Omron CX-Programmer project NewProject (CX-Programmer 9.75)

# PLC NewPLC1: CQM1 CPU43

## Program NewProgram1 (no task)

### Section Section1

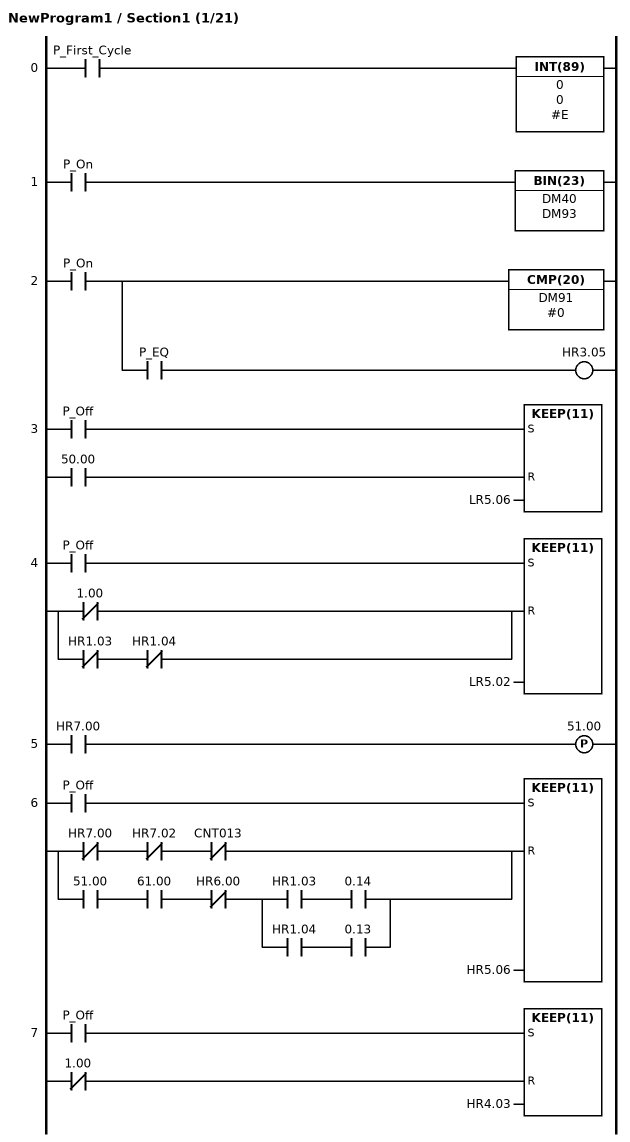
; rung 0
LD P_First_Cycle
INT(89) 0 0 #E
; rung 1
LD P_On
BIN(23) DM40 DM93
; rung 2
LD P_On
CMP(20) DM91 #0
AND P_EQ
OUT HR3.05
; rung 3
LD P_Off
LD 50.00
KEEP(11) LR5.06
; rung 4
LD P_Off
LDNOT 1.00
LDNOT HR1.03
ANDNOT HR1.04
ORLD
KEEP(11) LR5.02
; rung 5
LD HR7.00
DIFU(13) 51.00
; rung 6
LD P_Off
LDNOT HR7.00
ANDNOT HR7.02
ANDNOT CNT013
LD 51.00
AND 61.00
ANDNOT HR6.00
LD HR1.03
AND 0.14
LD HR1.04
AND 0.13
ORLD
ANDLD
ORLD
KEEP(11) HR5.06
; rung 7
LD P_Off
LDNOT 1.00
KEEP(11) HR4.03

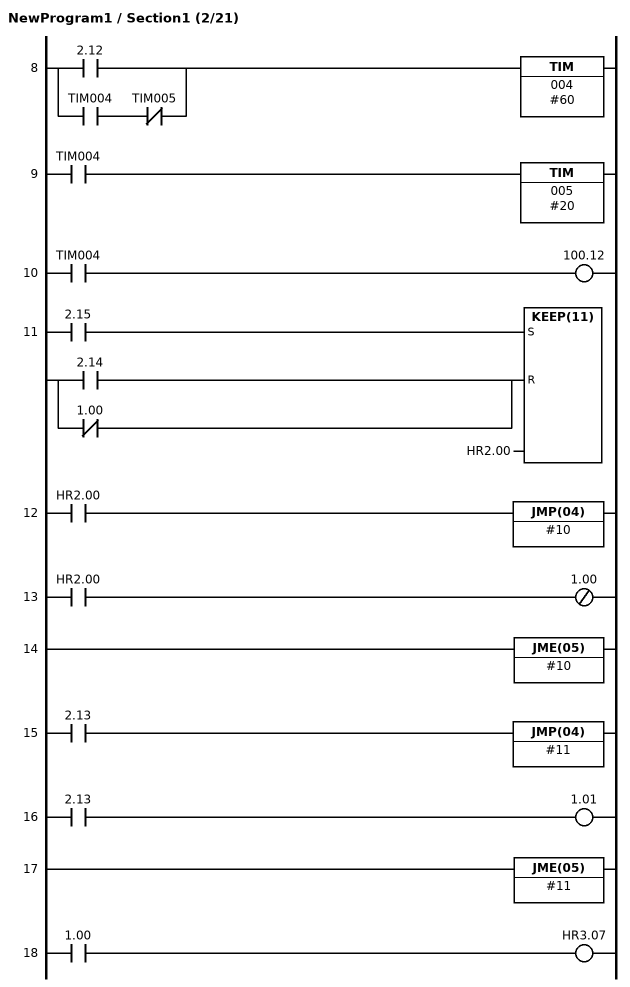
; rung 8
LD 2.12
LD TIM004
ANDNOT TIM005
ORLD
TIM 004 #60
; rung 9
LD TIM004
TIM 005 #20
; rung 10
LD TIM004
OUT 100.12
; rung 11
LD 2.15
LD 2.14
ORNOT 1.00
KEEP(11) HR2.00
; rung 12
LD HR2.00
JMP(04) #10
; rung 13
LD HR2.00
OUTNOT 1.00
; rung 14
JME(05) #10
; rung 15
LD 2.13
JMP(04) #11
; rung 16
LD 2.13
OUT 1.01
; rung 17
JME(05) #11
; rung 18
LD 1.00
OUT HR3.07

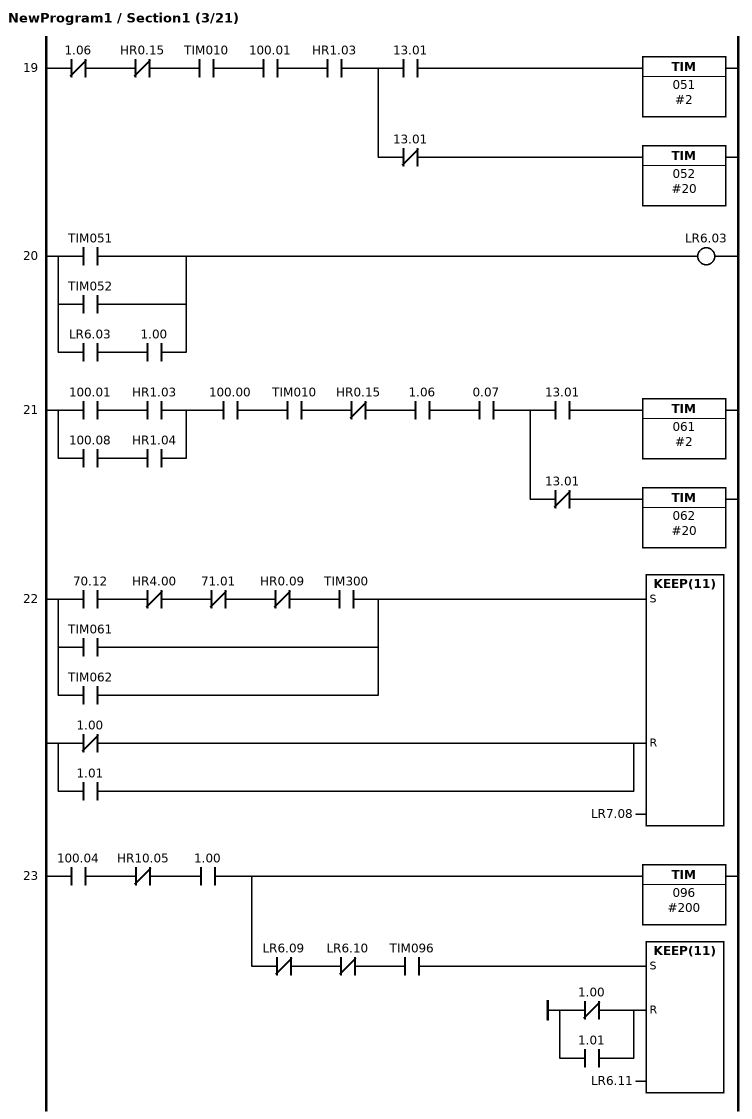
; rung 19
LDNOT 1.06
ANDNOT HR0.15
AND TIM010
AND 100.01
AND HR1.03
OUT TR0
AND 13.01
TIM 051 #2
LD TR0
ANDNOT 13.01
TIM 052 #20
; rung 20
LD TIM051
OR TIM052
LD LR6.03
AND 1.00
ORLD
OUT LR6.03
; rung 21
LD 100.01
AND HR1.03
LD 100.08
AND HR1.04
ORLD
AND 100.00
AND TIM010
ANDNOT HR0.15
AND 1.06
AND 0.07
OUT TR0
AND 13.01
TIM 061 #2
LD TR0
ANDNOT 13.01
TIM 062 #20
; rung 22
LD 70.12
ANDNOT HR4.00
ANDNOT 71.01
ANDNOT HR0.09
AND TIM300
OR TIM061
OR TIM062
LDNOT 1.00
OR 1.01
KEEP(11) LR7.08
; rung 23
LD 100.04
ANDNOT HR10.05
AND 1.00
TIM 096 #200
ANDNOT LR6.09
ANDNOT LR6.10
AND TIM096
LDNOT 1.00
OR 1.01
KEEP(11) LR6.11

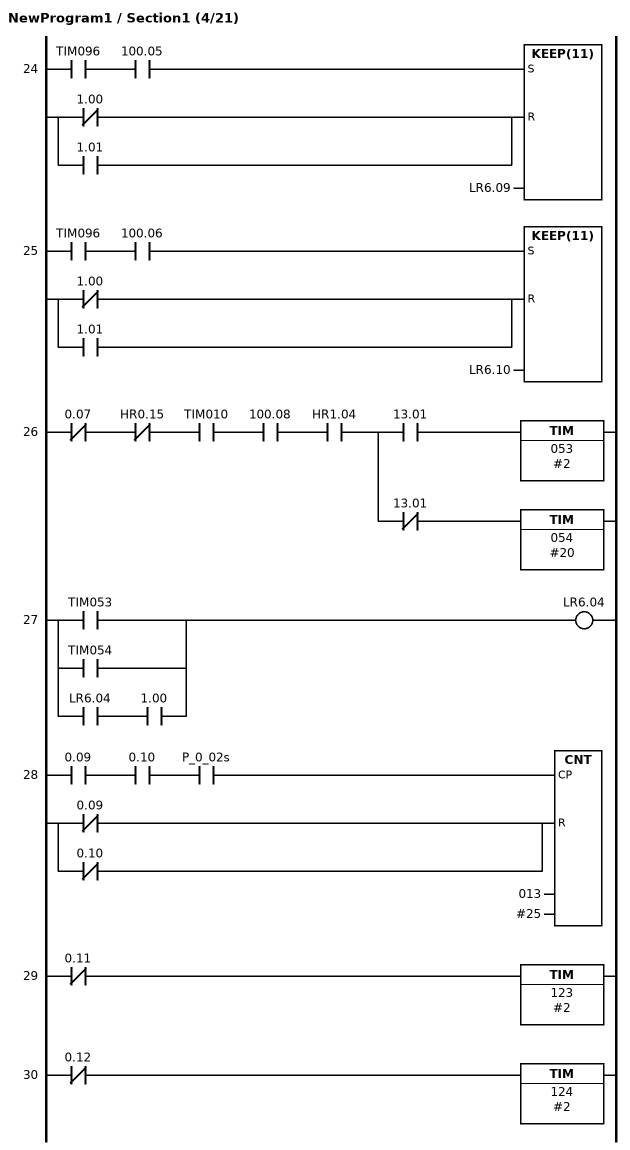
; rung 24
LD TIM096
AND 100.05
LDNOT 1.00
OR 1.01
KEEP(11) LR6.09
; rung 25
LD TIM096
AND 100.06
LDNOT 1.00
OR 1.01
KEEP(11) LR6.10
; rung 26
LDNOT 0.07
ANDNOT HR0.15
AND TIM010
AND 100.08
AND HR1.04
OUT TR0
AND 13.01
TIM 053 #2
LD TR0
ANDNOT 13.01
TIM 054 #20
; rung 27
LD TIM053
OR TIM054
LD LR6.04
AND 1.00
ORLD
OUT LR6.04
; rung 28
LD 0.09
AND 0.10
AND P_0_02s
LDNOT 0.09
ORNOT 0.10
CNT 013 #25
; rung 29
LDNOT 0.11
TIM 123 #2
; rung 30
LDNOT 0.12
TIM 124 #2

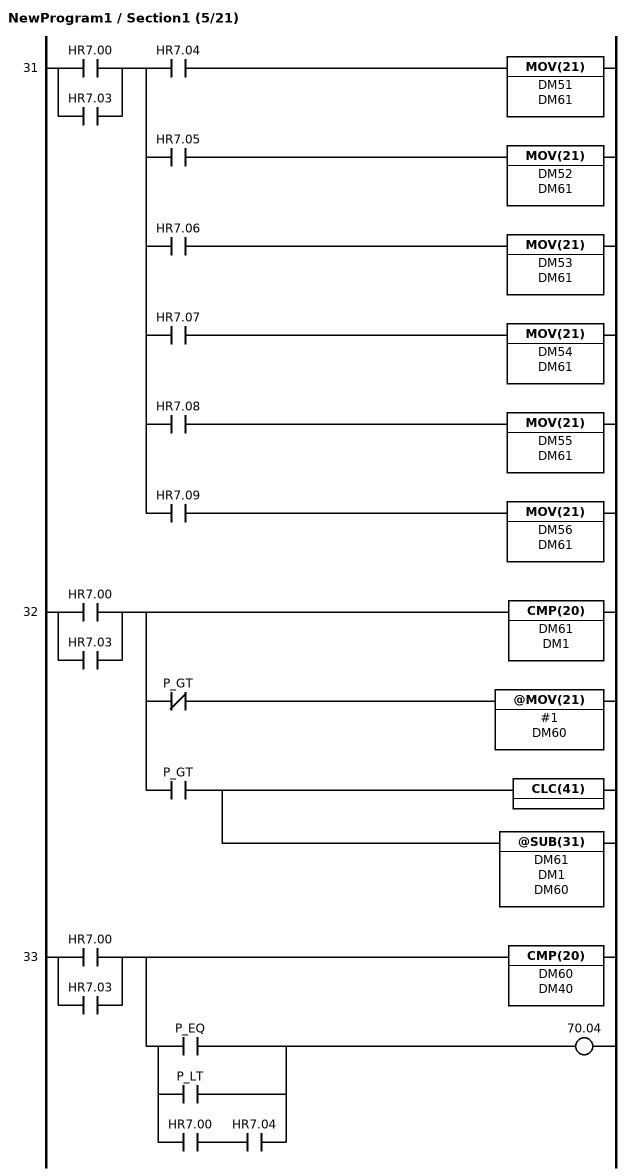
; rung 31
LD HR7.00
OR HR7.03
OUT TR0
AND HR7.04
MOV(21) DM51 DM61
LD TR0
AND HR7.05
MOV(21) DM52 DM61
LD TR0
AND HR7.06
MOV(21) DM53 DM61
LD TR0
AND HR7.07
MOV(21) DM54 DM61
LD TR0
AND HR7.08
MOV(21) DM55 DM61
LD TR0
AND HR7.09
MOV(21) DM56 DM61
; rung 32
LD HR7.00
OR HR7.03
OUT TR0
CMP(20) DM61 DM1
ANDNOT P_GT
@MOV(21) #1 DM60
LD TR0
AND P_GT
CLC(41)
@SUB(31) DM61 DM1 DM60
; rung 33
LD HR7.00
OR HR7.03
CMP(20) DM60 DM40
LD P_EQ
OR P_LT
LD HR7.00
AND HR7.04
ORLD
ANDLD
OUT 70.04

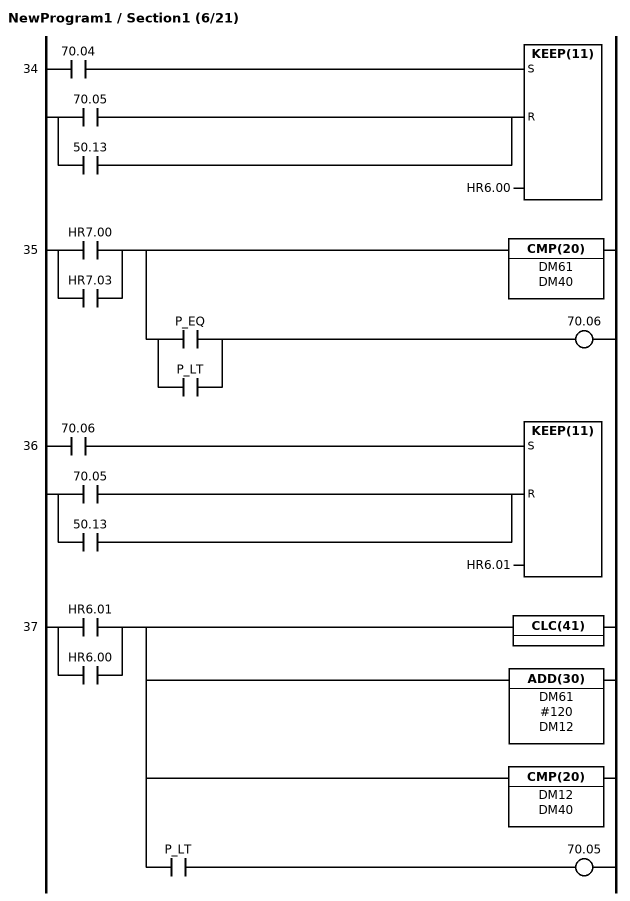
; rung 34
LD 70.04
LD 70.05
OR 50.13
KEEP(11) HR6.00
; rung 35
LD HR7.00
OR HR7.03
CMP(20) DM61 DM40
LD P_EQ
OR P_LT
ANDLD
OUT 70.06
; rung 36
LD 70.06
LD 70.05
OR 50.13
KEEP(11) HR6.01
; rung 37
LD HR6.01
OR HR6.00
CLC(41)
ADD(30) DM61 #120 DM12
CMP(20) DM12 DM40
AND P_LT
OUT 70.05

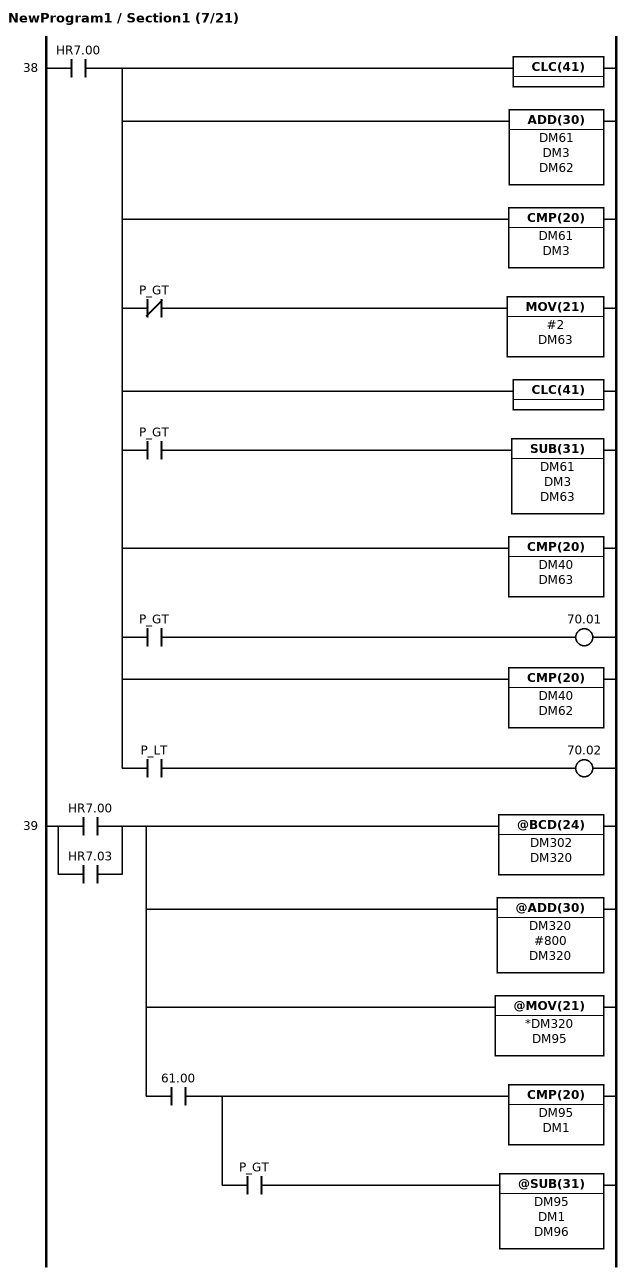
; rung 38
LD HR7.00
OUT TR0
CLC(41)
ADD(30) DM61 DM3 DM62
CMP(20) DM61 DM3
ANDNOT P_GT
MOV(21) #2 DM63
LD TR0
CLC(41)
AND P_GT
SUB(31) DM61 DM3 DM63
LD TR0
CMP(20) DM40 DM63
AND P_GT
OUT 70.01
LD TR0
CMP(20) DM40 DM62
AND P_LT
OUT 70.02
; rung 39
LD HR7.00
OR HR7.03
@BCD(24) DM302 DM320
@ADD(30) DM320 #800 DM320
@MOV(21) *DM320 DM95
AND 61.00
CMP(20) DM95 DM1
AND P_GT
@SUB(31) DM95 DM1 DM96

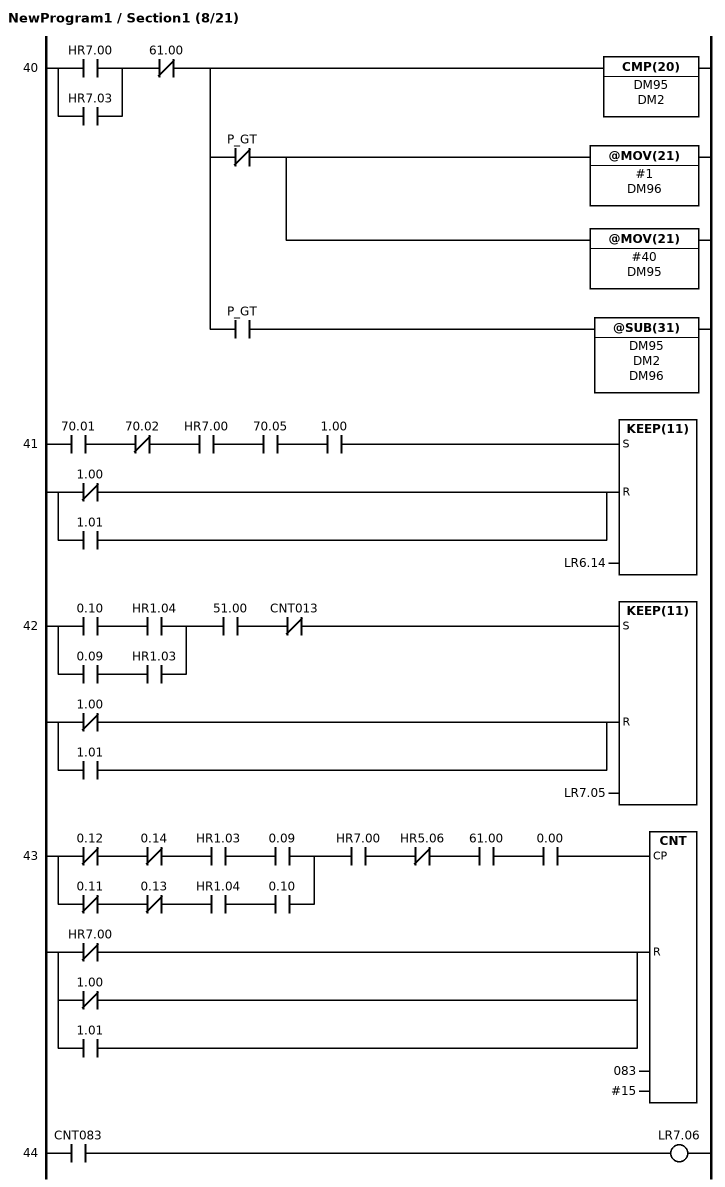
; rung 40
LD HR7.00
OR HR7.03
ANDNOT 61.00
OUT TR0
CMP(20) DM95 DM2
ANDNOT P_GT
@MOV(21) #1 DM96
@MOV(21) #40 DM95
LD TR0
AND P_GT
@SUB(31) DM95 DM2 DM96
; rung 41
LD 70.01
ANDNOT 70.02
AND HR7.00
AND 70.05
AND 1.00
LDNOT 1.00
OR 1.01
KEEP(11) LR6.14
; rung 42
LD 0.10
AND HR1.04
LD 0.09
AND HR1.03
ORLD
AND 51.00
ANDNOT CNT013
LDNOT 1.00
OR 1.01
KEEP(11) LR7.05
; rung 43
LDNOT 0.12
ANDNOT 0.14
AND HR1.03
AND 0.09
LDNOT 0.11
ANDNOT 0.13
AND HR1.04
AND 0.10
ORLD
AND HR7.00
ANDNOT HR5.06
AND 61.00
AND 0.00
LDNOT HR7.00
ORNOT 1.00
OR 1.01
CNT 083 #15
; rung 44
LD CNT083
OUT LR7.06

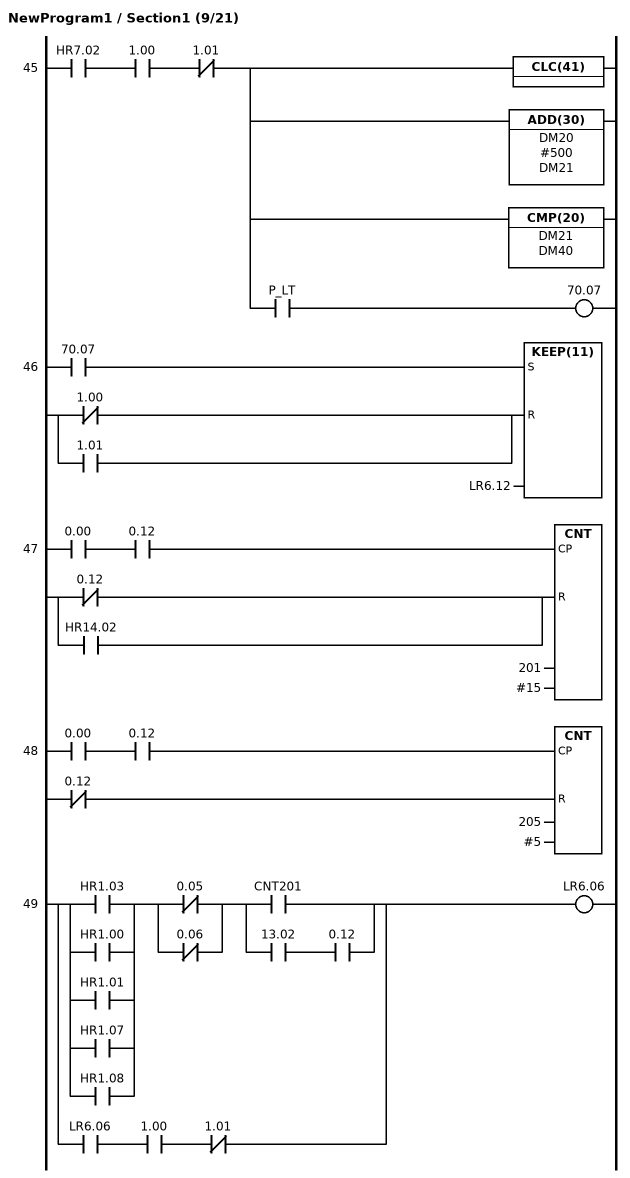
; rung 45
LD HR7.02
AND 1.00
ANDNOT 1.01
CLC(41)
ADD(30) DM20 #500 DM21
CMP(20) DM21 DM40
AND P_LT
OUT 70.07
; rung 46
LD 70.07
LDNOT 1.00
OR 1.01
KEEP(11) LR6.12
; rung 47
LD 0.00
AND 0.12
LDNOT 0.12
OR HR14.02
CNT 201 #15
; rung 48
LD 0.00
AND 0.12
LDNOT 0.12
CNT 205 #5
; rung 49
LD HR1.03
OR HR1.00
OR HR1.01
OR HR1.07
OR HR1.08
LDNOT 0.05
ORNOT 0.06
ANDLD
LD CNT201
LD 13.02
AND 0.12
ORLD
ANDLD
LD LR6.06
AND 1.00
ANDNOT 1.01
ORLD
OUT LR6.06

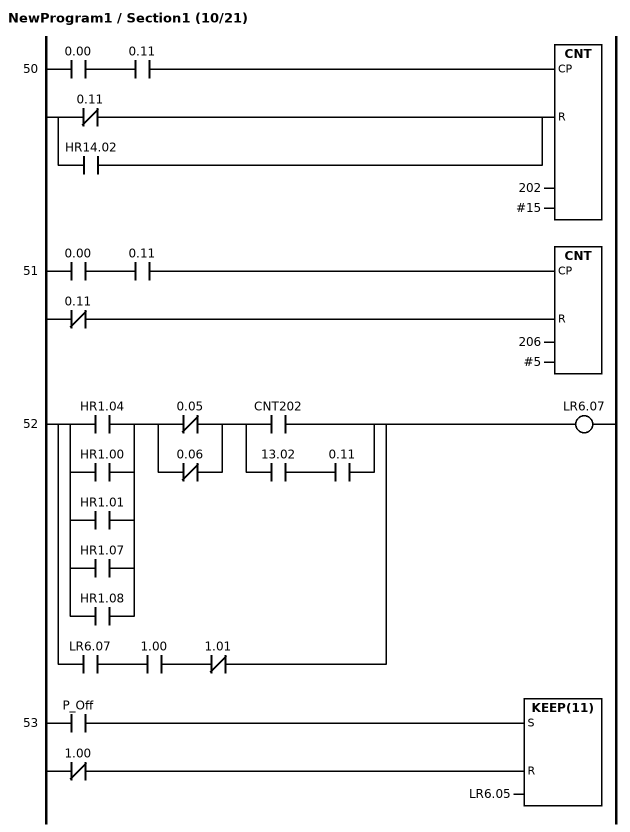
; rung 50
LD 0.00
AND 0.11
LDNOT 0.11
OR HR14.02
CNT 202 #15
; rung 51
LD 0.00
AND 0.11
LDNOT 0.11
CNT 206 #5
; rung 52
LD HR1.04
OR HR1.00
OR HR1.01
OR HR1.07
OR HR1.08
LDNOT 0.05
ORNOT 0.06
ANDLD
LD CNT202
LD 13.02
AND 0.11
ORLD
ANDLD
LD LR6.07
AND 1.00
ANDNOT 1.01
ORLD
OUT LR6.07
; rung 53
LD P_Off
LDNOT 1.00
KEEP(11) LR6.05

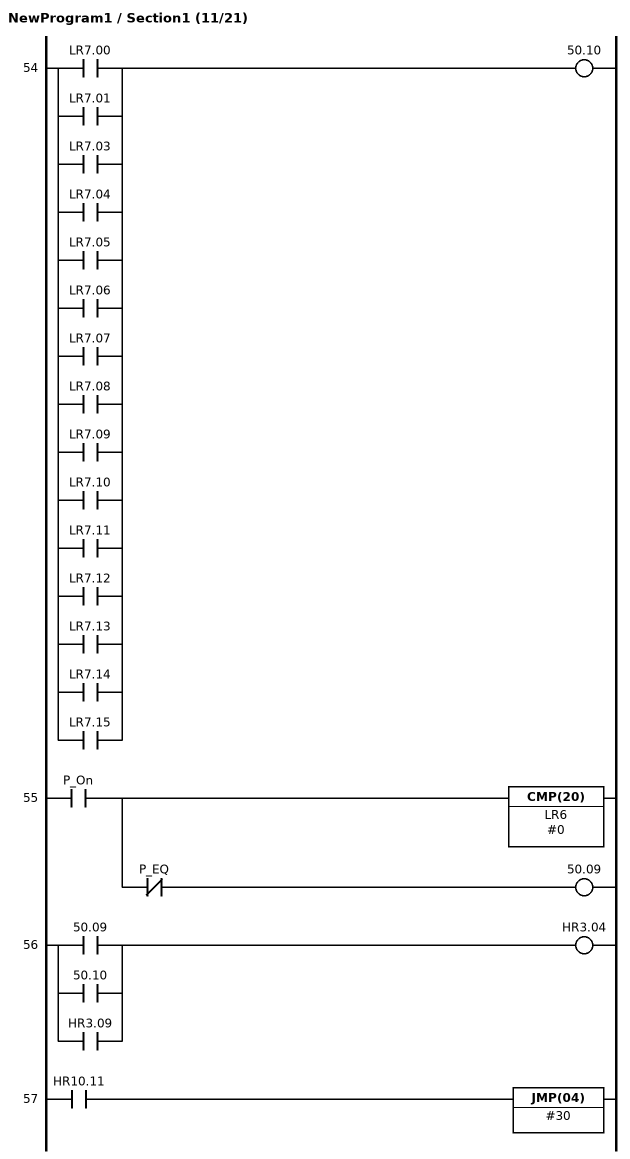
; rung 54
LD LR7.00
OR LR7.01
OR LR7.03
OR LR7.04
OR LR7.05
OR LR7.06
OR LR7.07
OR LR7.08
OR LR7.09
OR LR7.10
OR LR7.11
OR LR7.12
OR LR7.13
OR LR7.14
OR LR7.15
OUT 50.10
; rung 55
LD P_On
CMP(20) LR6 #0
ANDNOT P_EQ
OUT 50.09
; rung 56
LD 50.09
OR 50.10
OR HR3.09
OUT HR3.04
; rung 57
LD HR10.11
JMP(04) #30

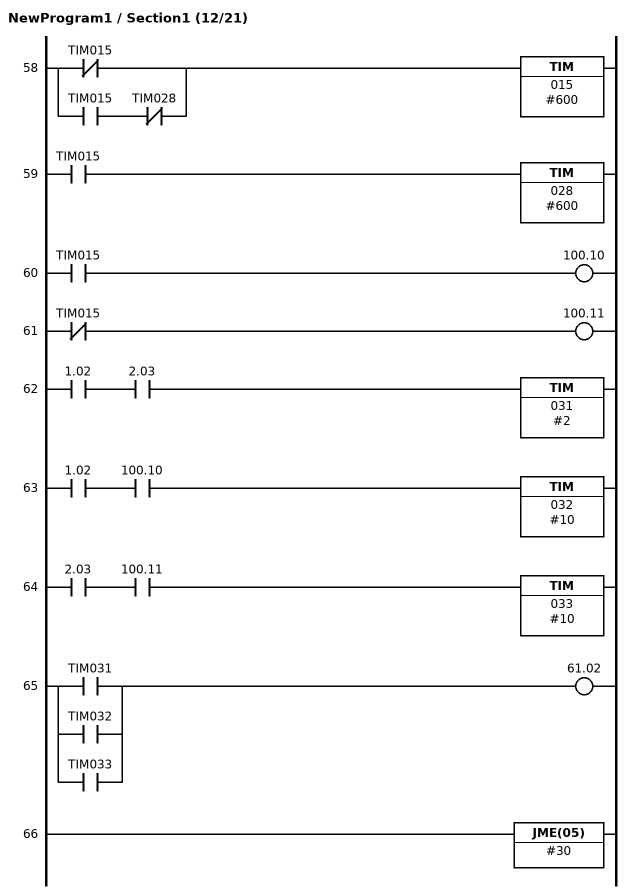
; rung 58
LDNOT TIM015
LD TIM015
ANDNOT TIM028
ORLD
TIM 015 #600
; rung 59
LD TIM015
TIM 028 #600
; rung 60
LD TIM015
OUT 100.10
; rung 61
LDNOT TIM015
OUT 100.11
; rung 62
LD 1.02
AND 2.03
TIM 031 #2
; rung 63
LD 1.02
AND 100.10
TIM 032 #10
; rung 64
LD 2.03
AND 100.11
TIM 033 #10
; rung 65
LD TIM031
OR TIM032
OR TIM033
OUT 61.02
; rung 66
JME(05) #30

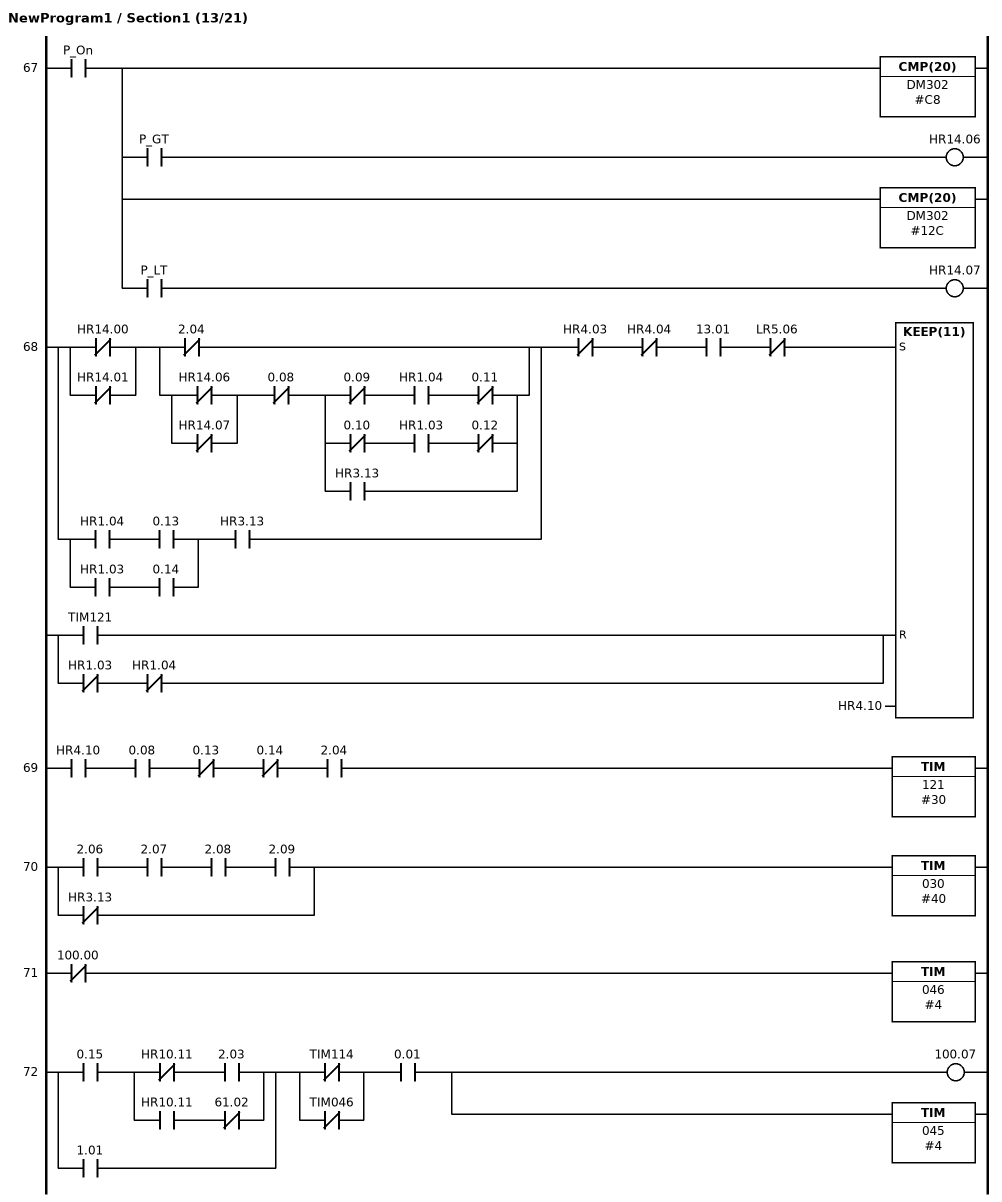
; rung 67
LD P_On
OUT TR0
CMP(20) DM302 #C8
AND P_GT
OUT HR14.06
LD TR0
CMP(20) DM302 #12C
AND P_LT
OUT HR14.07
; rung 68
LDNOT HR14.00
ORNOT HR14.01
LDNOT 2.04
LDNOT HR14.06
ORNOT HR14.07
ANDNOT 0.08
LDNOT 0.09
AND HR1.04
ANDNOT 0.11
LDNOT 0.10
AND HR1.03
ANDNOT 0.12
ORLD
OR HR3.13
ANDLD
ORLD
ANDLD
LD HR1.04
AND 0.13
LD HR1.03
AND 0.14
ORLD
AND HR3.13
ORLD
ANDNOT HR4.03
ANDNOT HR4.04
AND 13.01
ANDNOT LR5.06
LD TIM121
LDNOT HR1.03
ANDNOT HR1.04
ORLD
KEEP(11) HR4.10
; rung 69
LD HR4.10
AND 0.08
ANDNOT 0.13
ANDNOT 0.14
AND 2.04
TIM 121 #30
; rung 70
LD 2.06
AND 2.07
AND 2.08
AND 2.09
ORNOT HR3.13
TIM 030 #40
; rung 71
LDNOT 100.00
TIM 046 #4
; rung 72
LD 0.15
LDNOT HR10.11
AND 2.03
LD HR10.11
ANDNOT 61.02
ORLD
ANDLD
OR 1.01
LDNOT TIM114
ORNOT TIM046
ANDLD
AND 0.01
OUT 100.07
TIM 045 #4

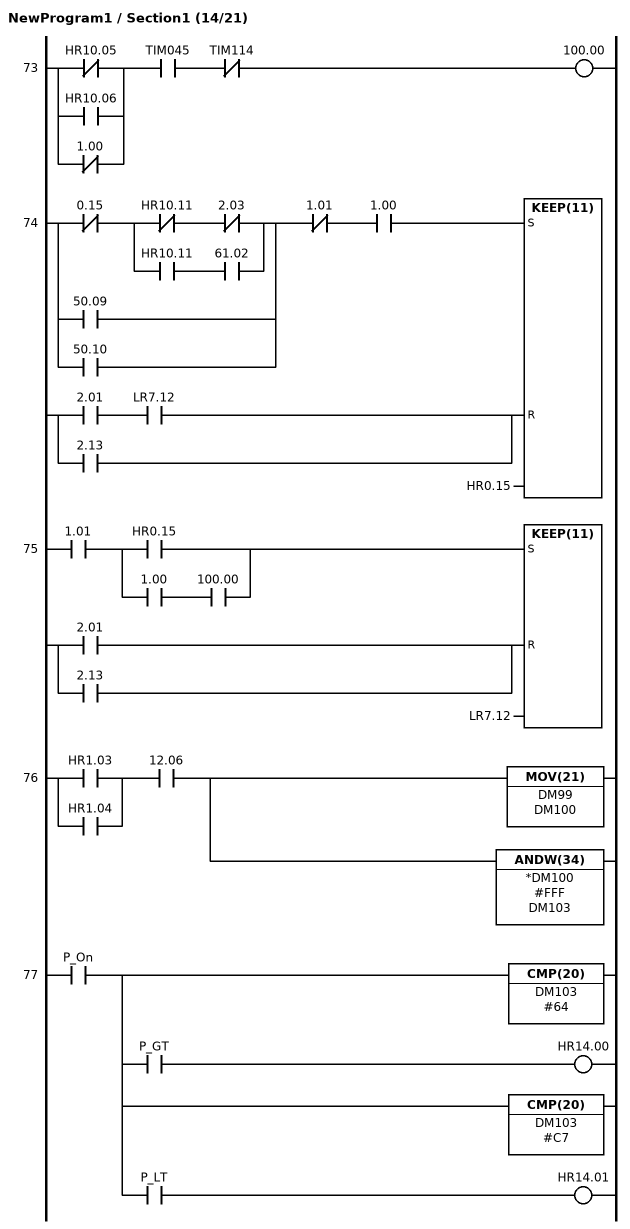
; rung 73
LDNOT HR10.05
OR HR10.06
ORNOT 1.00
AND TIM045
ANDNOT TIM114
OUT 100.00
; rung 74
LDNOT 0.15
LDNOT HR10.11
ANDNOT 2.03
LD HR10.11
AND 61.02
ORLD
ANDLD
OR 50.09
OR 50.10
ANDNOT 1.01
AND 1.00
LD 2.01
AND LR7.12
OR 2.13
KEEP(11) HR0.15
; rung 75
LD 1.01
LD HR0.15
LD 1.00
AND 100.00
ORLD
ANDLD
LD 2.01
OR 2.13
KEEP(11) LR7.12
; rung 76
LD HR1.03
OR HR1.04
AND 12.06
MOV(21) DM99 DM100
ANDW(34) *DM100 #FFF DM103
; rung 77
LD P_On
OUT TR0
CMP(20) DM103 #64
AND P_GT
OUT HR14.00
LD TR0
CMP(20) DM103 #C7
AND P_LT
OUT HR14.01

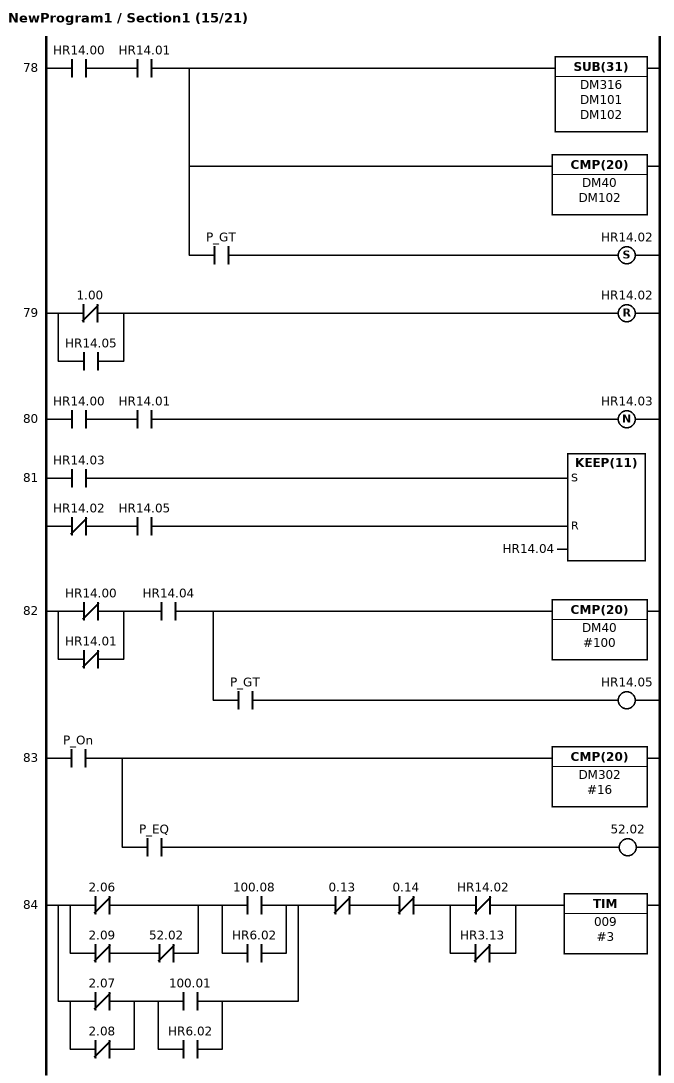
; rung 78
LD HR14.00
AND HR14.01
SUB(31) DM316 DM101 DM102
CMP(20) DM40 DM102
AND P_GT
SET HR14.02
; rung 79
LDNOT 1.00
OR HR14.05
RSET HR14.02
; rung 80
LD HR14.00
AND HR14.01
DIFD(14) HR14.03
; rung 81
LD HR14.03
LDNOT HR14.02
AND HR14.05
KEEP(11) HR14.04
; rung 82
LDNOT HR14.00
ORNOT HR14.01
AND HR14.04
CMP(20) DM40 #100
AND P_GT
OUT HR14.05
; rung 83
LD P_On
CMP(20) DM302 #16
AND P_EQ
OUT 52.02
; rung 84
LDNOT 2.06
LDNOT 2.09
ANDNOT 52.02
ORLD
LD 100.08
OR HR6.02
ANDLD
LDNOT 2.07
ORNOT 2.08
LD 100.01
OR HR6.02
ANDLD
ORLD
ANDNOT 0.13
ANDNOT 0.14
LDNOT HR14.02
ORNOT HR3.13
ANDLD
TIM 009 #3

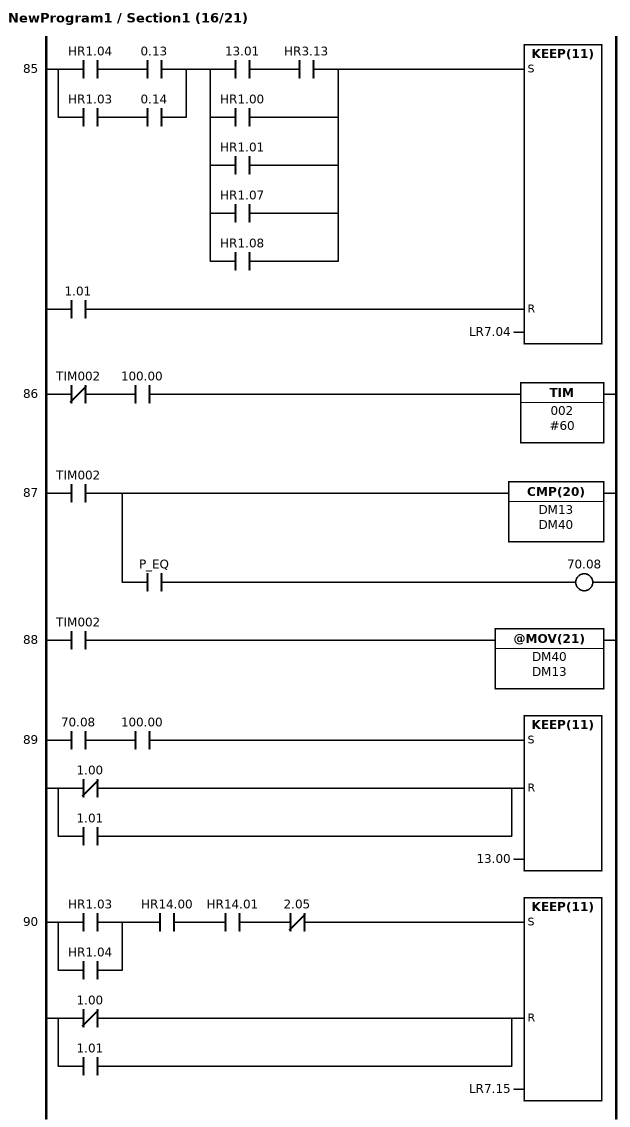
; rung 85
LD HR1.04
AND 0.13
LD HR1.03
AND 0.14
ORLD
LD 13.01
AND HR3.13
OR HR1.00
OR HR1.01
OR HR1.07
OR HR1.08
ANDLD
LD 1.01
KEEP(11) LR7.04
; rung 86
LDNOT TIM002
AND 100.00
TIM 002 #60
; rung 87
LD TIM002
CMP(20) DM13 DM40
AND P_EQ
OUT 70.08
; rung 88
LD TIM002
@MOV(21) DM40 DM13
; rung 89
LD 70.08
AND 100.00
LDNOT 1.00
OR 1.01
KEEP(11) 13.00
; rung 90
LD HR1.03
OR HR1.04
AND HR14.00
AND HR14.01
ANDNOT 2.05
LDNOT 1.00
OR 1.01
KEEP(11) LR7.15

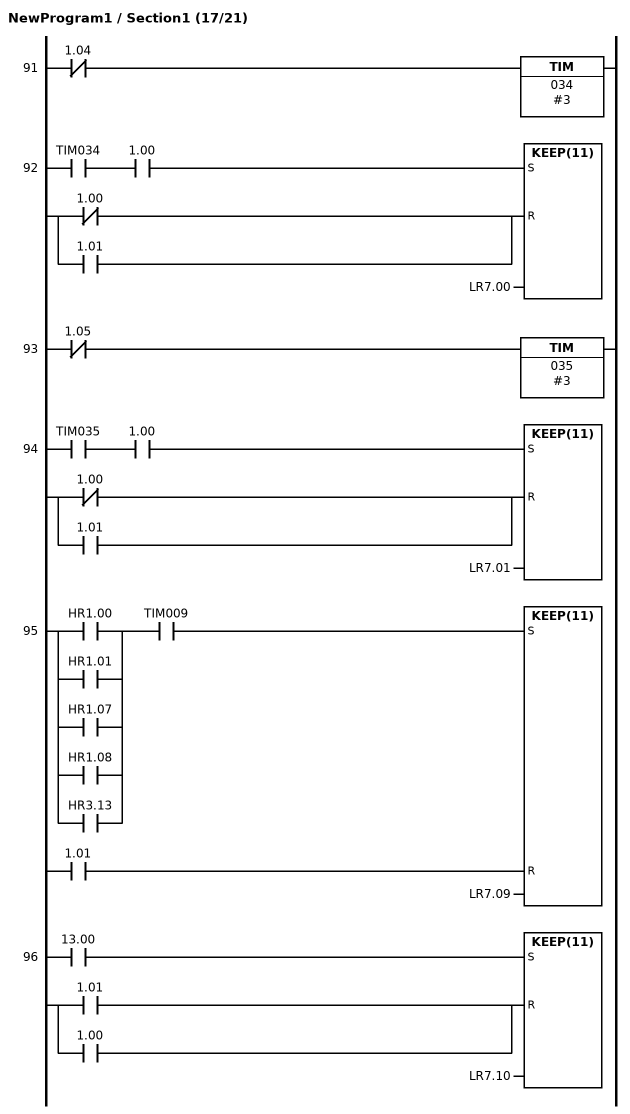
; rung 91
LDNOT 1.04
TIM 034 #3
; rung 92
LD TIM034
AND 1.00
LDNOT 1.00
OR 1.01
KEEP(11) LR7.00
; rung 93
LDNOT 1.05
TIM 035 #3
; rung 94
LD TIM035
AND 1.00
LDNOT 1.00
OR 1.01
KEEP(11) LR7.01
; rung 95
LD HR1.00
OR HR1.01
OR HR1.07
OR HR1.08
OR HR3.13
AND TIM009
LD 1.01
KEEP(11) LR7.09
; rung 96
LD 13.00
LD 1.01
OR 1.00
KEEP(11) LR7.10

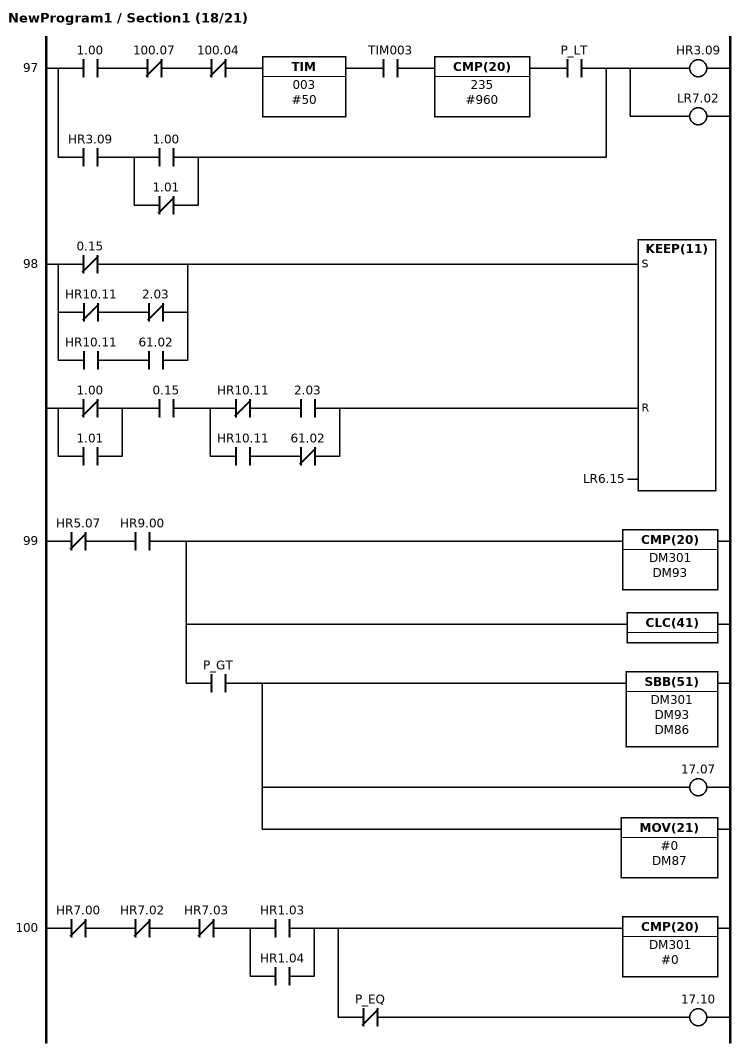
; rung 97
LD 1.00
ANDNOT 100.07
ANDNOT 100.04
TIM 003 #50
AND TIM003
CMP(20) 235 #960
AND P_LT
LD HR3.09
LD 1.00
ORNOT 1.01
ANDLD
ORLD
OUT HR3.09
OUT LR7.02
; rung 98
LDNOT 0.15
LDNOT HR10.11
ANDNOT 2.03
ORLD
LD HR10.11
AND 61.02
ORLD
LDNOT 1.00
OR 1.01
AND 0.15
LDNOT HR10.11
AND 2.03
LD HR10.11
ANDNOT 61.02
ORLD
ANDLD
KEEP(11) LR6.15
; rung 99
LDNOT HR5.07
AND HR9.00
CMP(20) DM301 DM93
CLC(41)
AND P_GT
SBB(51) DM301 DM93 DM86
OUT 17.07
MOV(21) #0 DM87
; rung 100
LDNOT HR7.00
ANDNOT HR7.02
ANDNOT HR7.03
LD HR1.03
OR HR1.04
ANDLD
CMP(20) DM301 #0
ANDNOT P_EQ
OUT 17.10

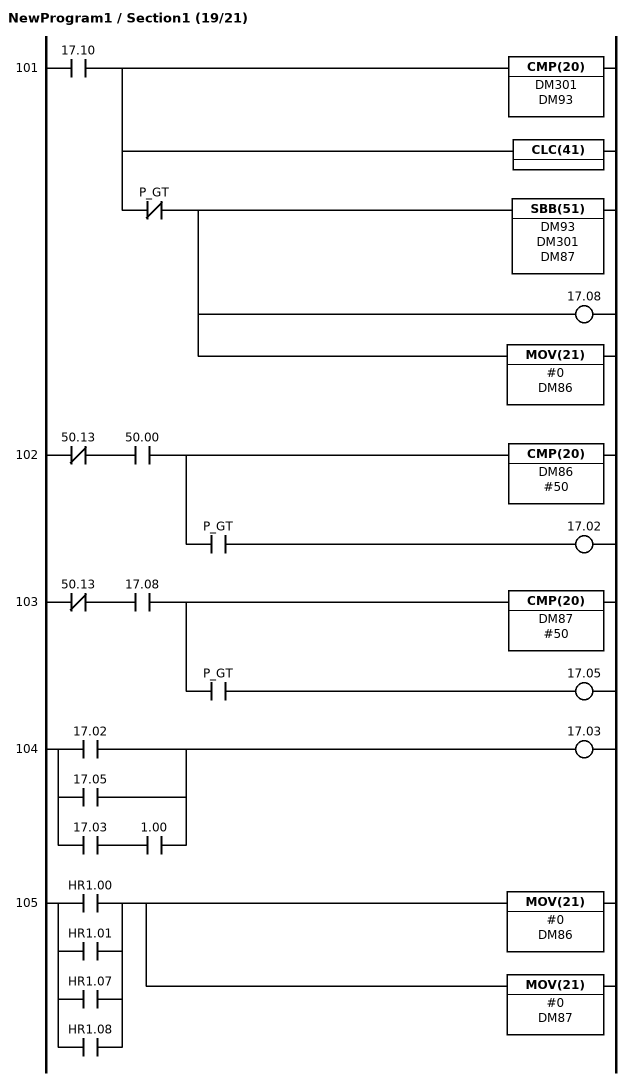
; rung 101
LD 17.10
CMP(20) DM301 DM93
CLC(41)
ANDNOT P_GT
SBB(51) DM93 DM301 DM87
OUT 17.08
MOV(21) #0 DM86
; rung 102
LDNOT 50.13
AND 50.00
CMP(20) DM86 #50
AND P_GT
OUT 17.02
; rung 103
LDNOT 50.13
AND 17.08
CMP(20) DM87 #50
AND P_GT
OUT 17.05
; rung 104
LD 17.02
OR 17.05
LD 17.03
AND 1.00
ORLD
OUT 17.03
; rung 105
LD HR1.00
OR HR1.01
OR HR1.07
OR HR1.08
MOV(21) #0 DM86
MOV(21) #0 DM87

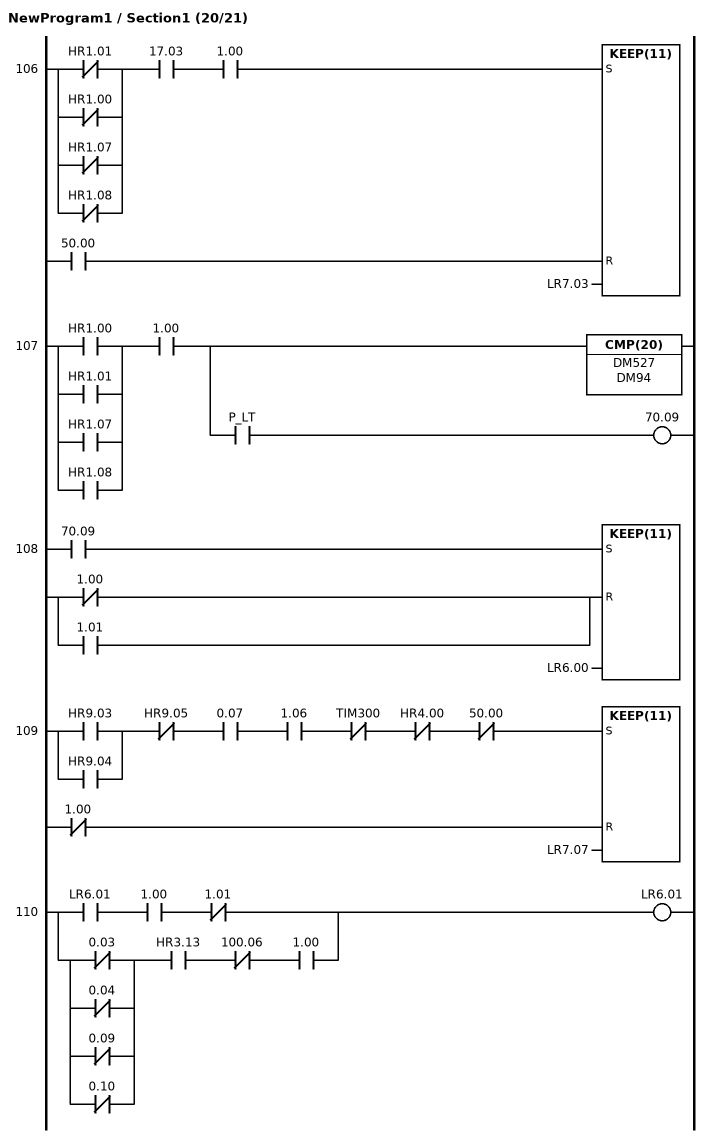
; rung 106
LDNOT HR1.01
ORNOT HR1.00
ORNOT HR1.07
ORNOT HR1.08
AND 17.03
AND 1.00
LD 50.00
KEEP(11) LR7.03
; rung 107
LD HR1.00
OR HR1.01
OR HR1.07
OR HR1.08
AND 1.00
CMP(20) DM527 DM94
AND P_LT
OUT 70.09
; rung 108
LD 70.09
LDNOT 1.00
OR 1.01
KEEP(11) LR6.00
; rung 109
LD HR9.03
OR HR9.04
ANDNOT HR9.05
AND 0.07
AND 1.06
ANDNOT TIM300
ANDNOT HR4.00
ANDNOT 50.00
LDNOT 1.00
KEEP(11) LR7.07
; rung 110
LD LR6.01
AND 1.00
ANDNOT 1.01
LDNOT 0.03
ORNOT 0.04
ORNOT 0.09
ORNOT 0.10
AND HR3.13
ANDNOT 100.06
AND 1.00
ORLD
OUT LR6.01

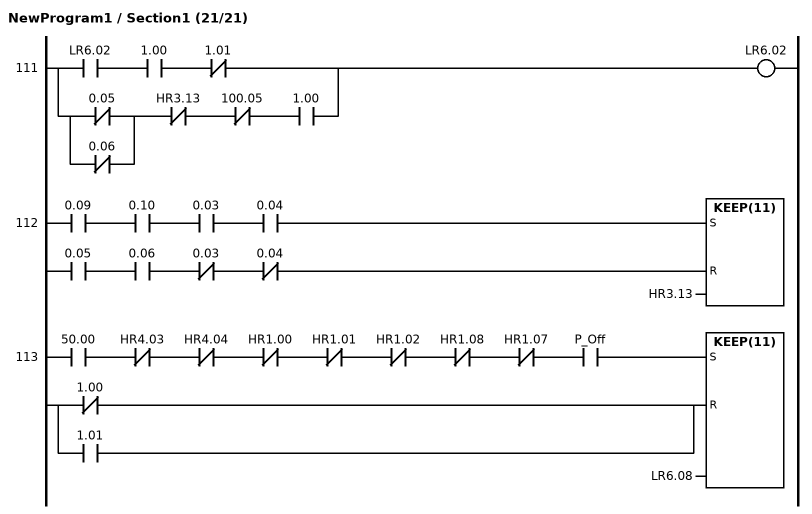
; rung 111
LD LR6.02
AND 1.00
ANDNOT 1.01
LDNOT 0.05
ORNOT 0.06
ANDNOT HR3.13
ANDNOT 100.05
AND 1.00
ORLD
OUT LR6.02
; rung 112
LD 0.09
AND 0.10
AND 0.03
AND 0.04
LD 0.05
AND 0.06
ANDNOT 0.03
ANDNOT 0.04
KEEP(11) HR3.13
; rung 113
LD 50.00
ANDNOT HR4.03
ANDNOT HR4.04
ANDNOT HR1.00
ANDNOT HR1.01
ANDNOT HR1.02
ANDNOT HR1.08
ANDNOT HR1.07
AND P_Off
LDNOT 1.00
OR 1.01
KEEP(11) LR6.08

### Section Section2

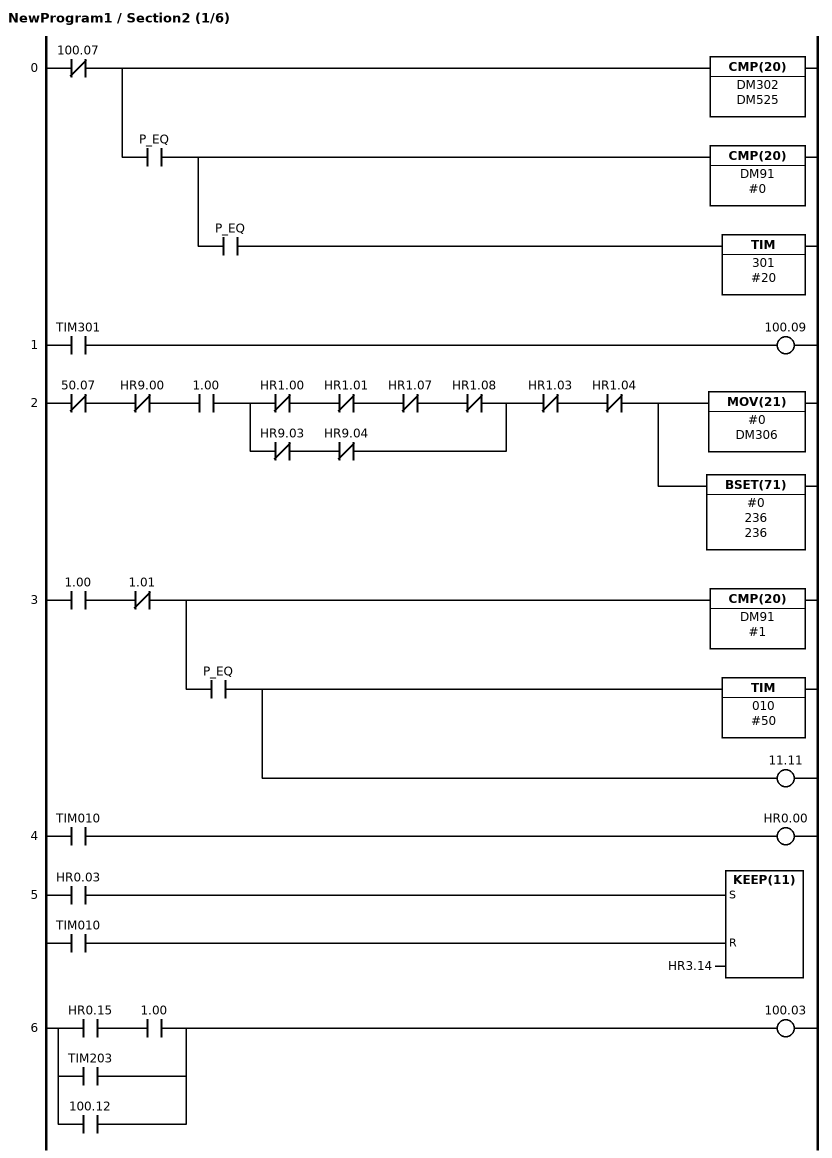
; rung 0
LDNOT 100.07
CMP(20) DM302 DM525
AND P_EQ
CMP(20) DM91 #0
AND P_EQ
TIM 301 #20
; rung 1
LD TIM301
OUT 100.09
; rung 2
LDNOT 50.07
ANDNOT HR9.00
AND 1.00
LDNOT HR1.00
ANDNOT HR1.01
ANDNOT HR1.07
ANDNOT HR1.08
LDNOT HR9.03
ANDNOT HR9.04
ORLD
ANDLD
ANDNOT HR1.03
ANDNOT HR1.04
MOV(21) #0 DM306
BSET(71) #0 236 236
; rung 3
LD 1.00
ANDNOT 1.01
CMP(20) DM91 #1
AND P_EQ
TIM 010 #50
OUT 11.11
; rung 4
LD TIM010
OUT HR0.00
; rung 5
LD HR0.03
LD TIM010
KEEP(11) HR3.14
; rung 6
LD HR0.15
AND 1.00
OR TIM203
OR 100.12
OUT 100.03

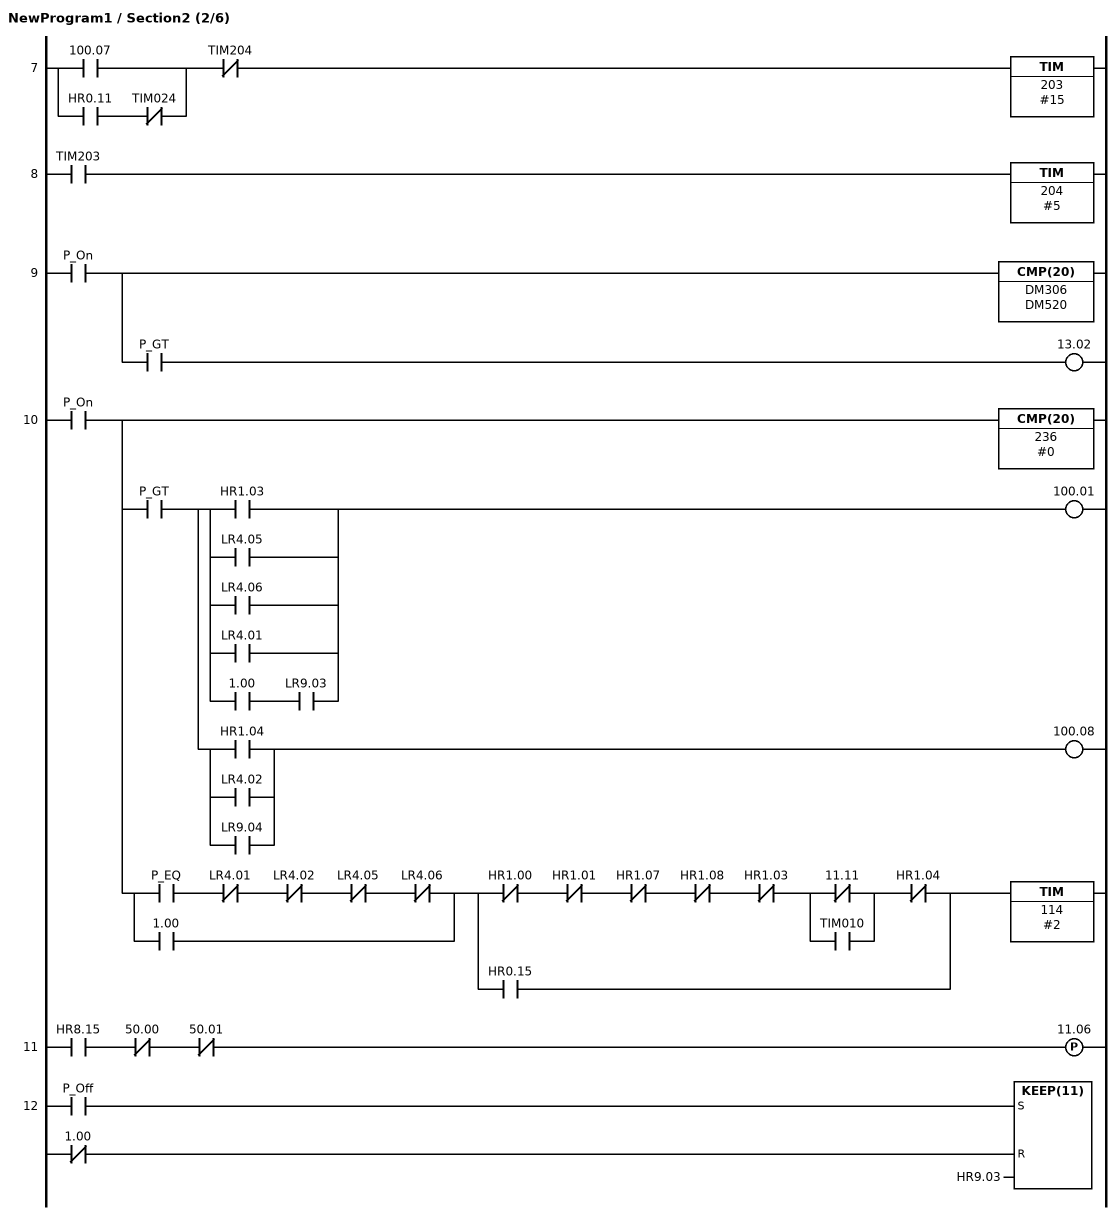
; rung 7
LD 100.07
LD HR0.11
ANDNOT TIM024
ORLD
ANDNOT TIM204
TIM 203 #15
; rung 8
LD TIM203
TIM 204 #5
; rung 9
LD P_On
CMP(20) DM306 DM520
AND P_GT
OUT 13.02
; rung 10
LD P_On
OUT TR0
CMP(20) 236 #0
AND P_GT
OUT TR1
LD HR1.03
OR LR4.05
OR LR4.06
OR LR4.01
LD 1.00
AND LR9.03
ORLD
ANDLD
OUT 100.01
LD TR1
LD HR1.04
OR LR4.02
OR LR9.04
ANDLD
OUT 100.08
LD TR0
LD P_EQ
ANDNOT LR4.01
ANDNOT LR4.02
ANDNOT LR4.05
ANDNOT LR4.06
OR 1.00
ANDLD
LDNOT HR1.00
ANDNOT HR1.01
ANDNOT HR1.07
ANDNOT HR1.08
ANDNOT HR1.03
LDNOT 11.11
OR TIM010
ANDLD
ANDNOT HR1.04
OR HR0.15
ANDLD
TIM 114 #2
; rung 11
LD HR8.15
ANDNOT 50.00
ANDNOT 50.01
DIFU(13) 11.06
; rung 12
LD P_Off
LDNOT 1.00
KEEP(11) HR9.03

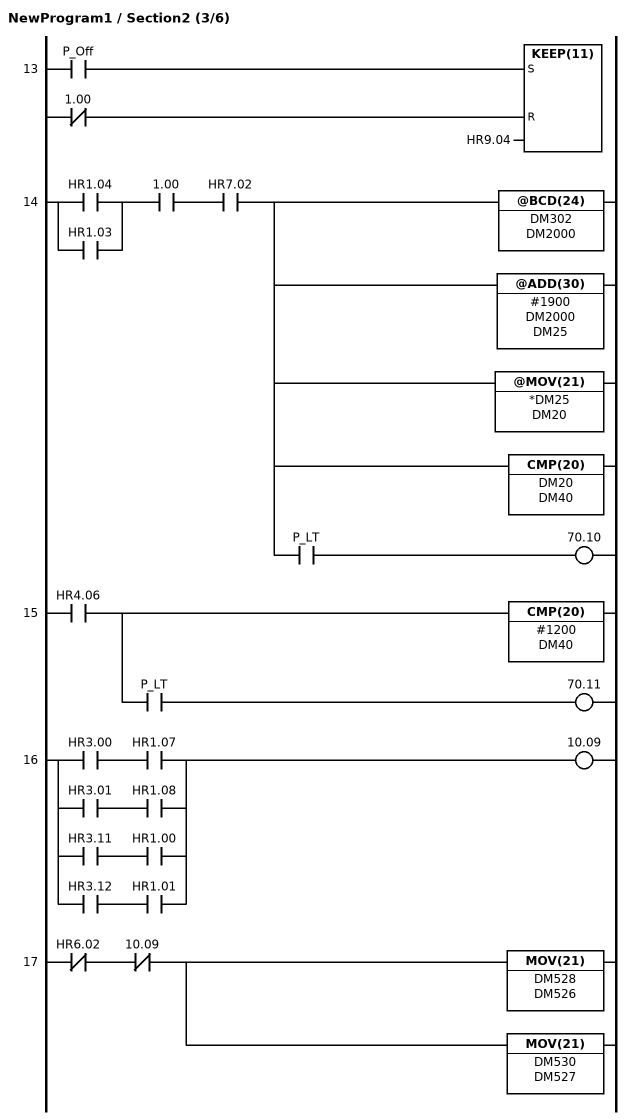
; rung 13
LD P_Off
LDNOT 1.00
KEEP(11) HR9.04
; rung 14
LD HR1.04
OR HR1.03
AND 1.00
AND HR7.02
@BCD(24) DM302 DM2000
@ADD(30) #1900 DM2000 DM25
@MOV(21) *DM25 DM20
CMP(20) DM20 DM40
AND P_LT
OUT 70.10
; rung 15
LD HR4.06
CMP(20) #1200 DM40
AND P_LT
OUT 70.11
; rung 16
LD HR3.00
AND HR1.07
LD HR3.01
AND HR1.08
ORLD
LD HR3.11
AND HR1.00
ORLD
LD HR3.12
AND HR1.01
ORLD
OUT 10.09
; rung 17
LDNOT HR6.02
ANDNOT 10.09
MOV(21) DM528 DM526
MOV(21) DM530 DM527

